(* Logix 5000 project; controller L3 vendor 1 type 14 code 92 rev 20.12; software revision 20.04; part 8 of 9 *)
(* tags used below, declared in another part *)
   A_CV_COLMAT : REAL;
   aux_spano : DINT;
   B3 : DINT[100];
   CONV_PID_N10_130 : PID;   // *** Tag created for conversion to PID type required for instruction translation ***
   CSG_N_VENTILO : REAL;
   CV_ANO : REAL;
   dif_I_red : DINT;
   F8 : REAL[100];
   inc_ano : DINT;
   khighano : DINT;
   klowano : DINT;
   L3_stat : DINT[20];
   limBBtano : DINT;
   limBtano : DINT;
   limhhtano : DINT;
   limhtano : DINT;
   M_nbr_ventilo_ano : DINT;
   mem_i_tot : DINT;
   N10 : DINT[233];
   N7 : DINT[200];
   N9 : DINT[200];   // niveau decapage vers lancy (n9[10) ;;N9[70]
   NCOM : INT[20];
   offsetano : DINT;
   offsetano_tdesc : DINT;
   offsetano_Tup : DINT;
   par_p1_ano : DINT;
   par_p2_ano : DINT;
   par_p3_ano : DINT;
   par_p4_ano : DINT;
   par_p5_ano : DINT;
   par_p6_ano : DINT;
   pid_ANO : PID;
   pid_colmat : PID;
   PIDwkk : PID;
   s_bp_neutral : BOOL;
   s_bp_stop_acide : BOOL;
   s_bp_strt_acide : BOOL;
   s_csg_ventilo_ano : DINT;
   s_nbr_ventilo_ano : DINT;
   S_Q_DEM_h2so4 : DINT;
   S_SP_ANO : DINT;
   S_T_ANO : DINT;
   SCP_CV_ANO : SCP;
   SCP_CV_COLMAT : SCP;
   SCP_CV_VENTILO : SCP;
   stat_L3 : DINT[20];
   T4 : TIMER[180];
   wkk_L3 : DINT[125];
(* _2_GENERAL, continued *)

ROUTINE _5_ACIDE   (* ladder *)
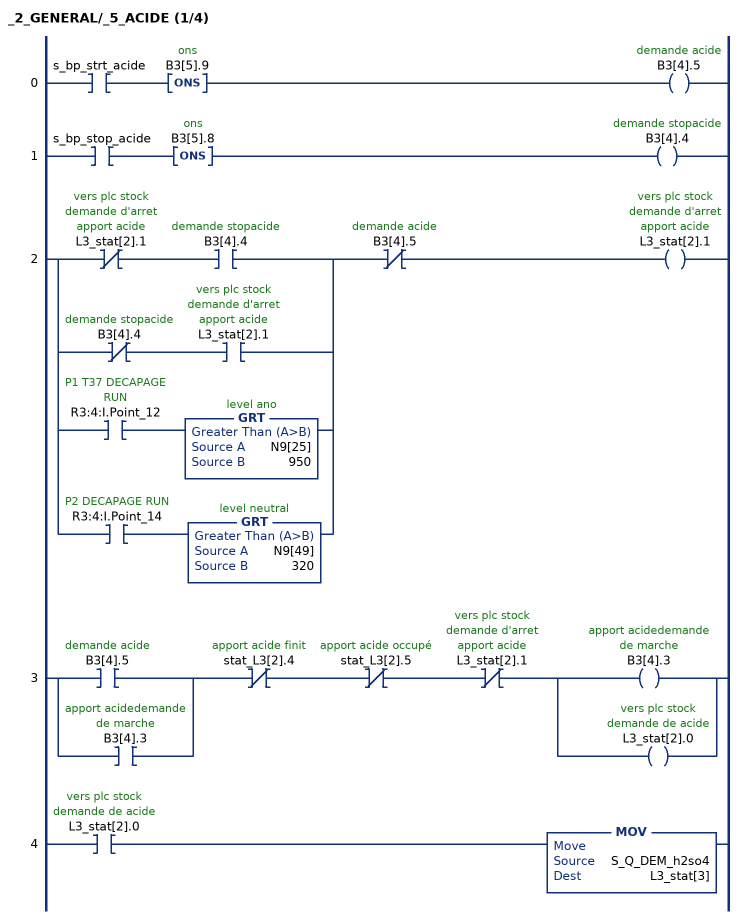
   0: XIC(s_bp_strt_acide)ONS(B3[5].9)OTE(B3[4].5);
   1: XIC(s_bp_stop_acide)ONS(B3[5].8)OTE(B3[4].4);
   2: [XIO(L3_stat[2].1) XIC(B3[4].4) ,XIO(B3[4].4) XIC(L3_stat[2].1) ,XIC(R3:4:I.Point_12) GRT(N9[25],950) ,XIC(R3:4:I.Point_14) GRT(N9[49],320) ]XIO(B3[4].5)OTE(L3_stat[2].1);
   3: [XIC(B3[4].5) ,XIC(B3[4].3) ]XIO(stat_L3[2].4)XIO(stat_L3[2].5)XIO(L3_stat[2].1)[OTE(B3[4].3) ,OTE(L3_stat[2].0) ];
   4: XIC(L3_stat[2].0)MOV(S_Q_DEM_h2so4,L3_stat[3]);
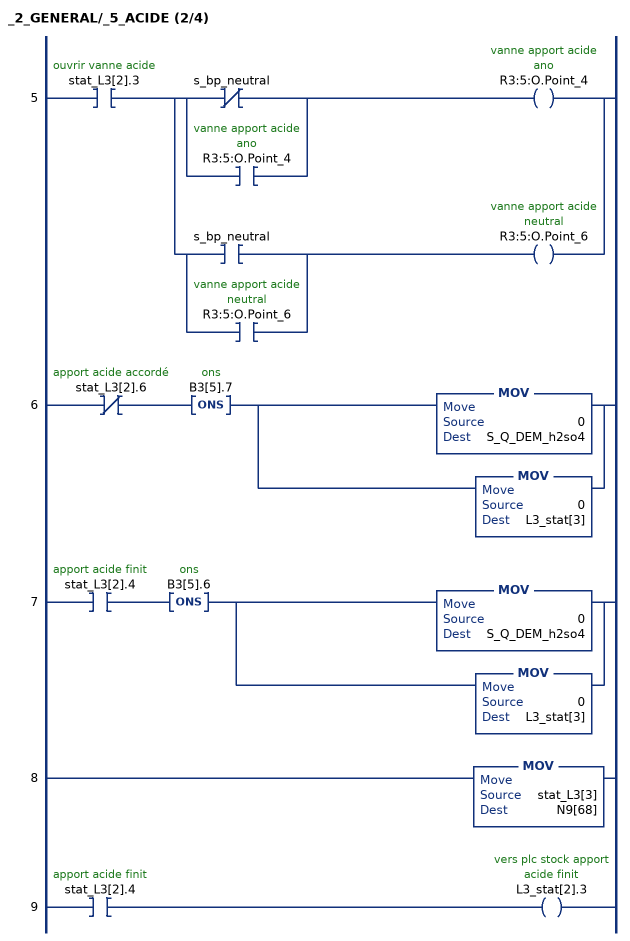
   5: XIC(stat_L3[2].3)[[XIO(s_bp_neutral) ,XIC(R3:5:O.Point_4) ] OTE(R3:5:O.Point_4) ,[XIC(s_bp_neutral) ,XIC(R3:5:O.Point_6) ] OTE(R3:5:O.Point_6) ];
   6: XIO(stat_L3[2].6)ONS(B3[5].7)[MOV(0,S_Q_DEM_h2so4) ,MOV(0,L3_stat[3]) ];
   7: XIC(stat_L3[2].4)ONS(B3[5].6)[MOV(0,S_Q_DEM_h2so4) ,MOV(0,L3_stat[3]) ];
   8: MOV(stat_L3[3],N9[68]);
   9: XIC(stat_L3[2].4)OTE(L3_stat[2].3);
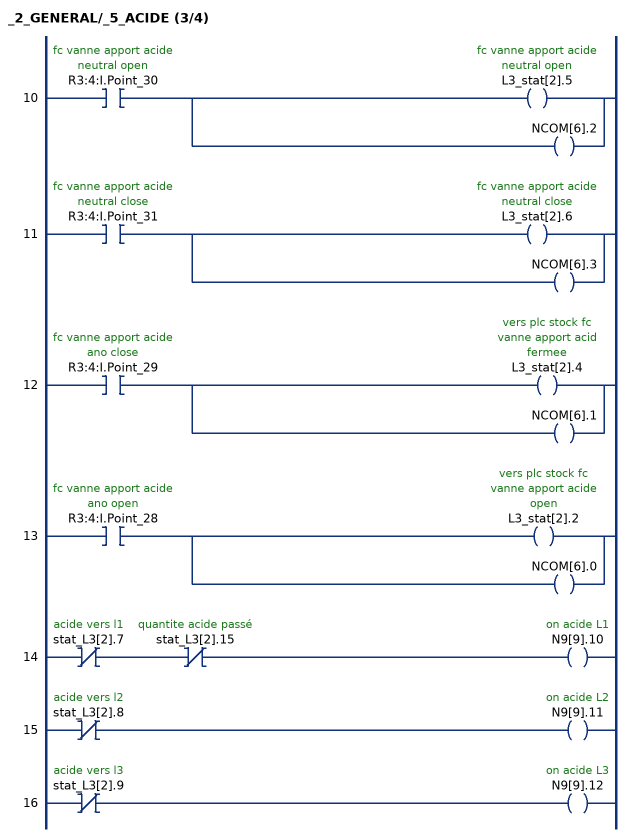
   10: XIC(R3:4:I.Point_30)[OTE(L3_stat[2].5) ,OTE(NCOM[6].2) ];
   11: XIC(R3:4:I.Point_31)[OTE(L3_stat[2].6) ,OTE(NCOM[6].3) ];
   12: XIC(R3:4:I.Point_29)[OTE(L3_stat[2].4) ,OTE(NCOM[6].1) ];
   13: XIC(R3:4:I.Point_28)[OTE(L3_stat[2].2) ,OTE(NCOM[6].0) ];
   14: XIO(stat_L3[2].7)XIO(stat_L3[2].15)OTE(N9[9].10);
   15: XIO(stat_L3[2].8)OTE(N9[9].11);
   16: XIO(stat_L3[2].9)OTE(N9[9].12);
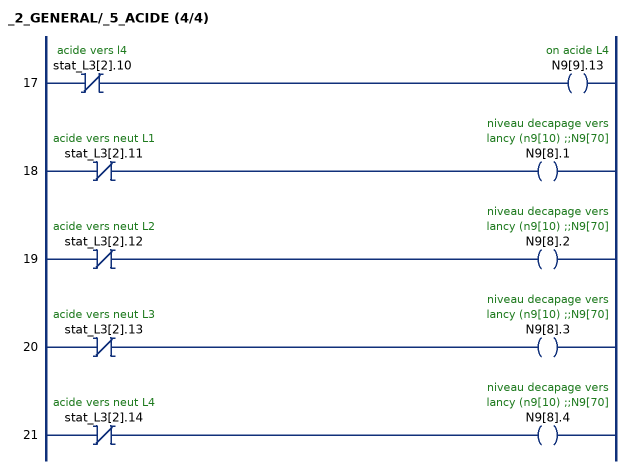
   17: XIO(stat_L3[2].10)OTE(N9[9].13);
   18: XIO(stat_L3[2].11)OTE(N9[8].1);
   19: XIO(stat_L3[2].12)OTE(N9[8].2);
   20: XIO(stat_L3[2].13)OTE(N9[8].3);
   21: XIO(stat_L3[2].14)OTE(N9[8].4);
END_ROUTINE

ROUTINE _6_REG_T_COL   (* ladder *)
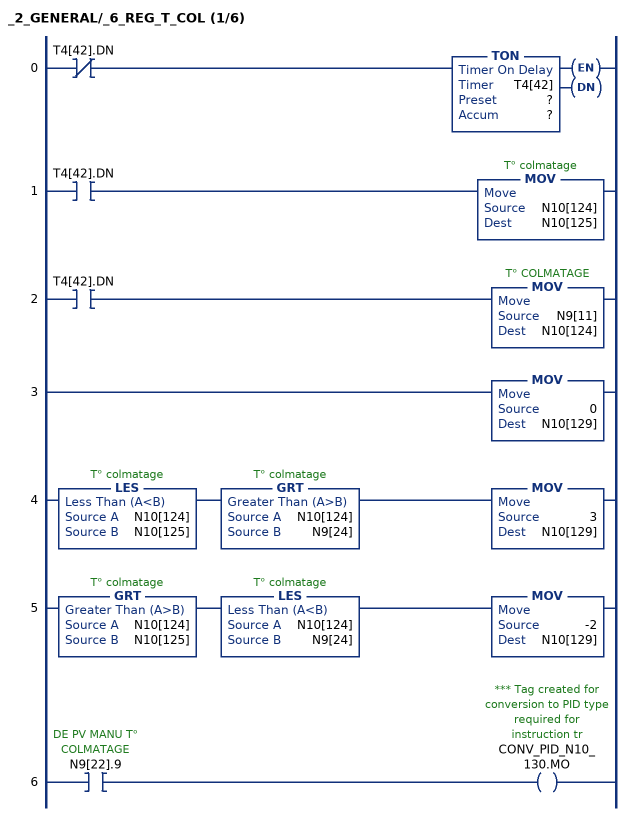
   0: XIO(T4[42].DN)TON(T4[42],?,?);
   1: XIC(T4[42].DN)MOV(N10[124],N10[125]);
   2: XIC(T4[42].DN)MOV(N9[11],N10[124]);
   3: MOV(0,N10[129]);
   4: LES(N10[124],N10[125])GRT(N10[124],N9[24])MOV(3,N10[129]);
   5: GRT(N10[124],N10[125])LES(N10[124],N9[24])MOV(-2,N10[129]);
   6: XIC(N9[22].9)OTE(CONV_PID_N10_130.MO);
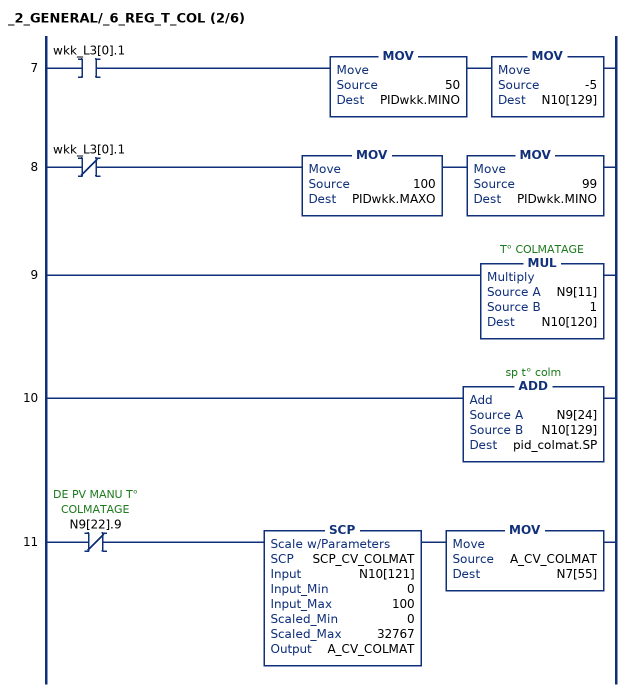
   7: XIC(wkk_L3[0].1)MOV(50,PIDwkk.MINO)MOV(-5,N10[129]);
   8: XIO(wkk_L3[0].1)MOV(100,PIDwkk.MAXO)MOV(99,PIDwkk.MINO);
   9: MUL(N9[11],1,N10[120]);
   10: ADD(N9[24],N10[129],pid_colmat.SP);
   11: XIO(N9[22].9)SCP(SCP_CV_COLMAT,N10[121],0,100,0,32767,A_CV_COLMAT)MOV(A_CV_COLMAT,N7[55]);
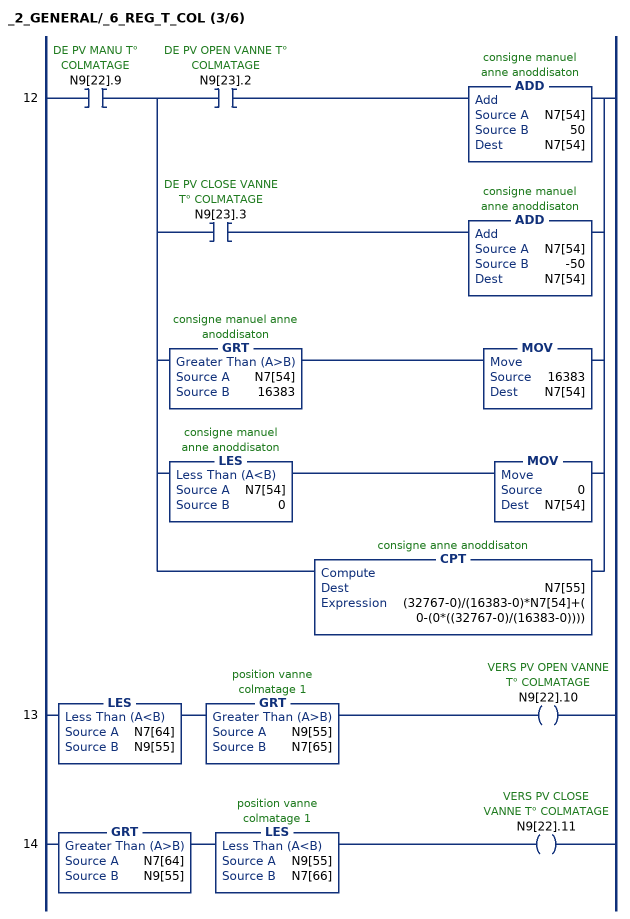
   12: XIC(N9[22].9)[XIC(N9[23].2) ADD(N7[54],50,N7[54]) ,XIC(N9[23].3) ADD(N7[54],-50,N7[54]) ,GRT(N7[54],16383) MOV(16383,N7[54]) ,LES(N7[54],0) MOV(0,N7[54]) ,CPT(N7[55],(32767-0)/(16383-0)*N7[54]+(0-(0*((32767-0)/(16383-0))))) ];
   13: LES(N7[64],N9[55])GRT(N9[55],N7[65])OTE(N9[22].10);
   14: GRT(N7[64],N9[55])LES(N9[55],N7[66])OTE(N9[22].11);
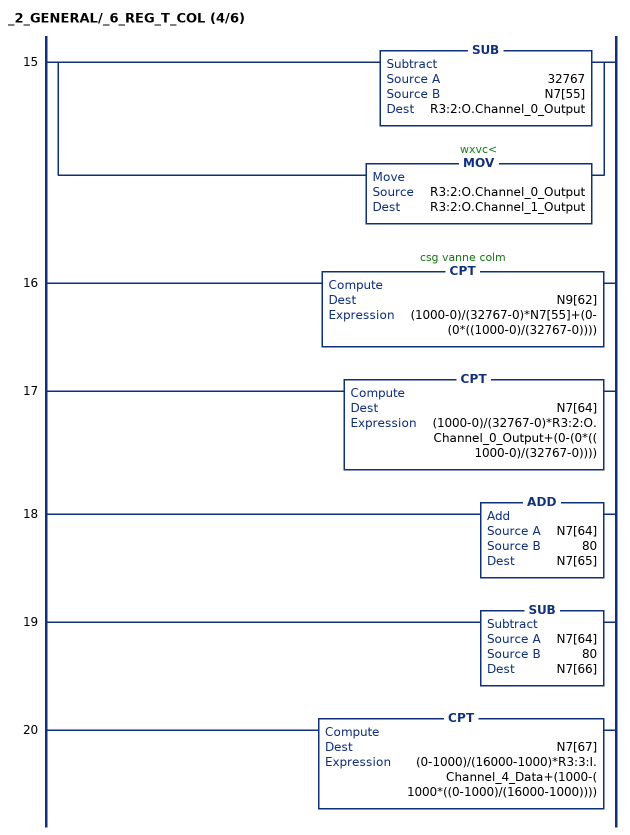
   15: [SUB(32767,N7[55],R3:2:O.Channel_0_Output) ,MOV(R3:2:O.Channel_0_Output,R3:2:O.Channel_1_Output) ];
   16: CPT(N9[62],(1000-0)/(32767-0)*N7[55]+(0-(0*((1000-0)/(32767-0)))));
   17: CPT(N7[64],(1000-0)/(32767-0)*R3:2:O.Channel_0_Output+(0-(0*((1000-0)/(32767-0)))));
   18: ADD(N7[64],80,N7[65]);
   19: SUB(N7[64],80,N7[66]);
   20: CPT(N7[67],(0-1000)/(16000-1000)*R3:3:I.Channel_4_Data+(1000-(1000*((0-1000)/(16000-1000)))));
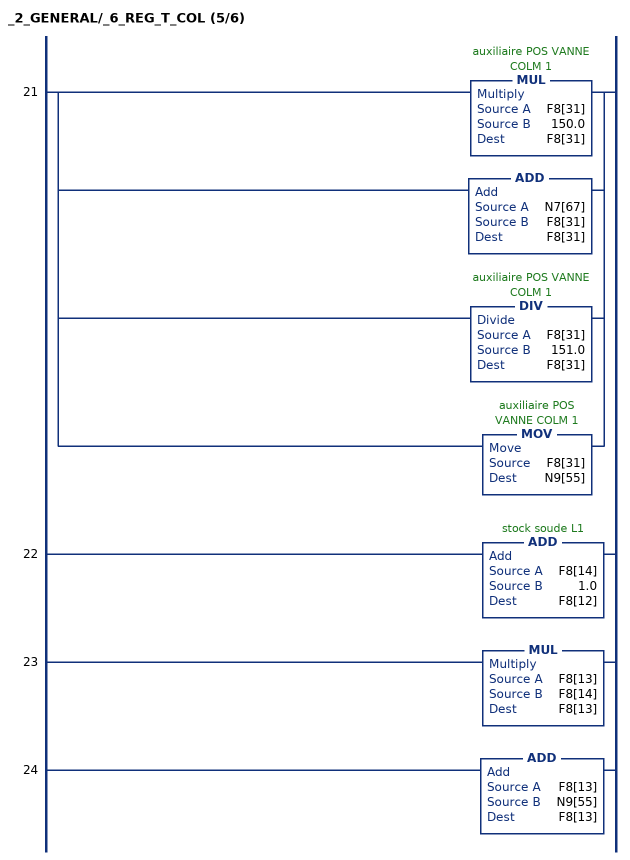
   21: [MUL(F8[31],150.0,F8[31]) ,ADD(N7[67],F8[31],F8[31]) ,DIV(F8[31],151.0,F8[31]) ,MOV(F8[31],N9[55]) ];
   22: ADD(F8[14],1.0,F8[12]);
   23: MUL(F8[13],F8[14],F8[13]);
   24: ADD(F8[13],N9[55],F8[13]);
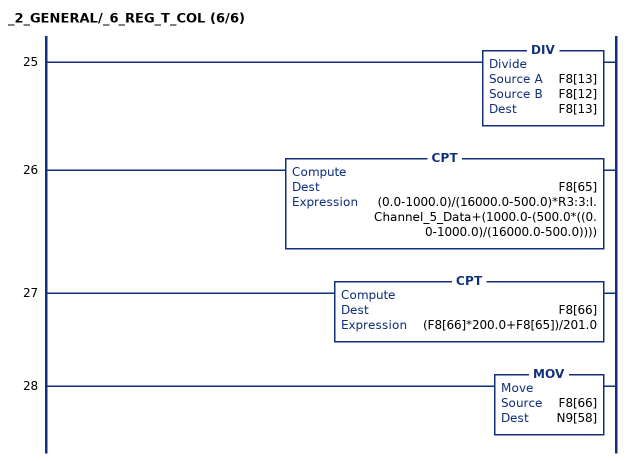
   25: DIV(F8[13],F8[12],F8[13]);
   26: CPT(F8[65],(0.0-1000.0)/(16000.0-500.0)*R3:3:I.Channel_5_Data+(1000.0-(500.0*((0.0-1000.0)/(16000.0-500.0)))));
   27: CPT(F8[66],(F8[66]*200.0+F8[65])/201.0);
   28: MOV(F8[66],N9[58]);
END_ROUTINE

ROUTINE _9_regul_ano   (* ladder *)
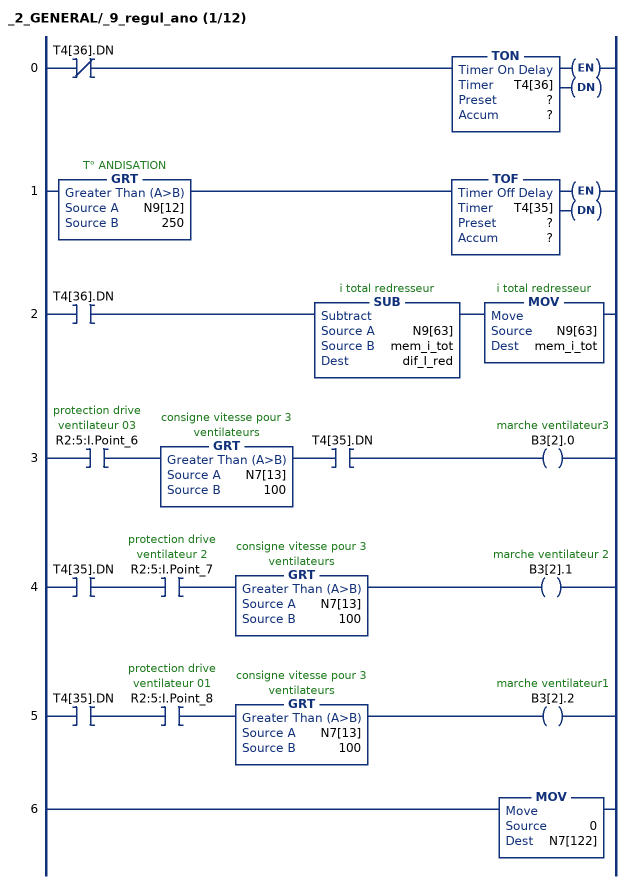
   0: XIO(T4[36].DN)TON(T4[36],?,?);
   1: GRT(N9[12],250)TOF(T4[35],?,?);
   2: XIC(T4[36].DN)SUB(N9[63],mem_i_tot,dif_I_red)MOV(N9[63],mem_i_tot);
   3: XIC(R2:5:I.Point_6)GRT(N7[13],100)XIC(T4[35].DN)OTE(B3[2].0);
   4: XIC(T4[35].DN)XIC(R2:5:I.Point_7)GRT(N7[13],100)OTE(B3[2].1);
   5: XIC(T4[35].DN)XIC(R2:5:I.Point_8)GRT(N7[13],100)OTE(B3[2].2);
   6: MOV(0,N7[122]);
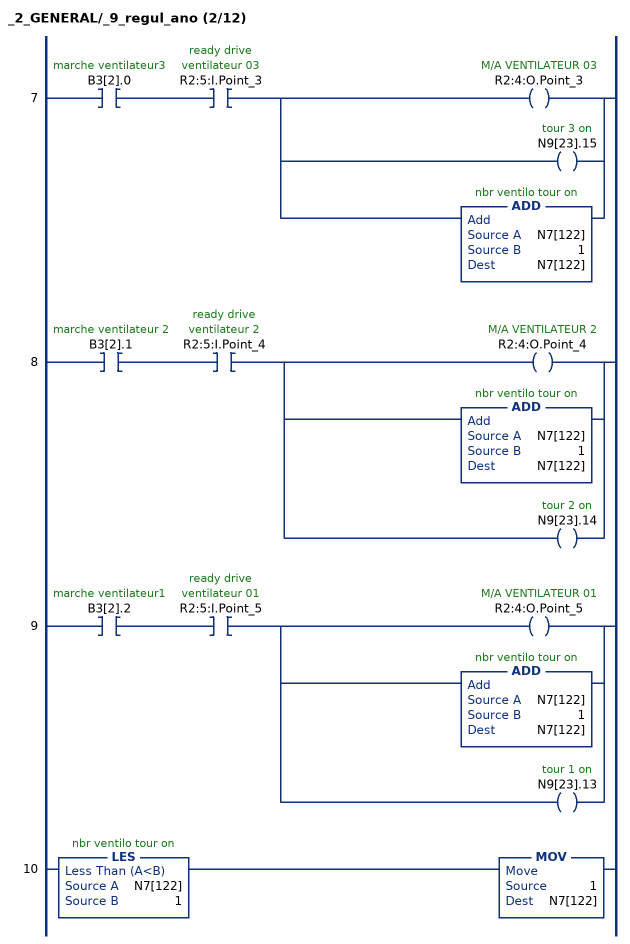
   7: XIC(B3[2].0)XIC(R2:5:I.Point_3)[OTE(R2:4:O.Point_3) ,OTE(N9[23].15) ,ADD(N7[122],1,N7[122]) ];
   8: XIC(B3[2].1)XIC(R2:5:I.Point_4)[OTE(R2:4:O.Point_4) ,ADD(N7[122],1,N7[122]) ,OTE(N9[23].14) ];
   9: XIC(B3[2].2)XIC(R2:5:I.Point_5)[OTE(R2:4:O.Point_5) ,ADD(N7[122],1,N7[122]) ,OTE(N9[23].13) ];
   10: LES(N7[122],1)MOV(1,N7[122]);
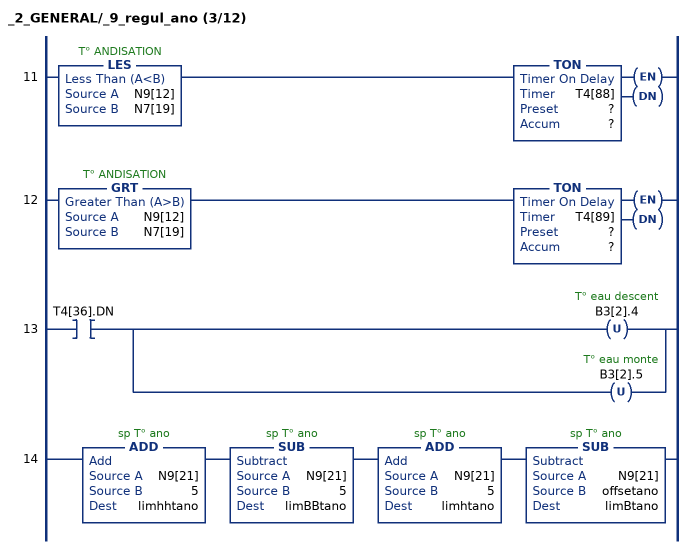
   11: LES(N9[12],N7[19])TON(T4[88],?,?);
   12: GRT(N9[12],N7[19])TON(T4[89],?,?);
   13: XIC(T4[36].DN)[OTU(B3[2].4) ,OTU(B3[2].5) ];
   14: ADD(N9[21],5,limhhtano)SUB(N9[21],5,limBBtano)ADD(N9[21],5,limhtano)SUB(N9[21],offsetano,limBtano);
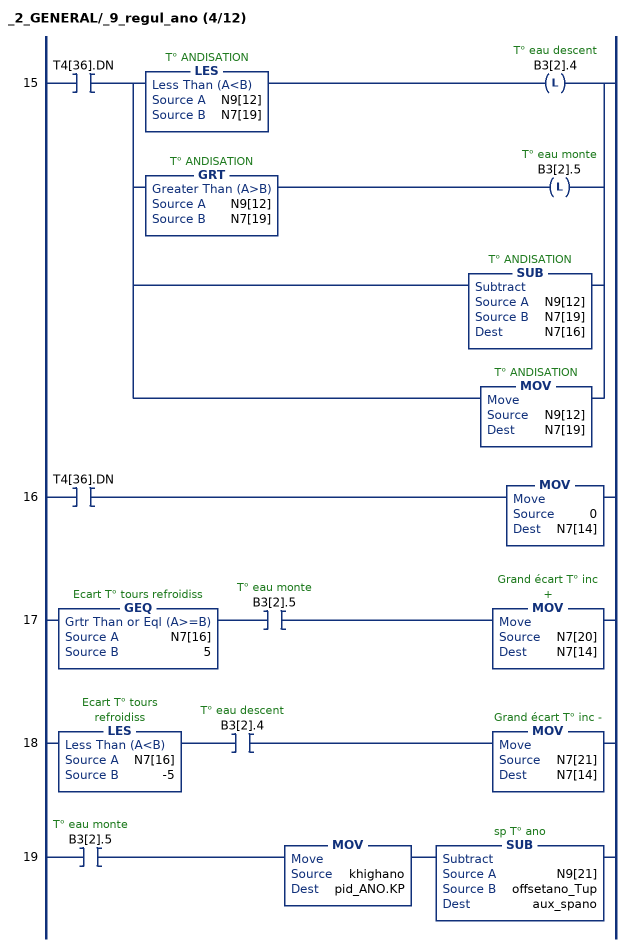
   15: XIC(T4[36].DN)[LES(N9[12],N7[19]) OTL(B3[2].4) ,GRT(N9[12],N7[19]) OTL(B3[2].5) ,SUB(N9[12],N7[19],N7[16]) ,MOV(N9[12],N7[19]) ];
   16: XIC(T4[36].DN)MOV(0,N7[14]);
   17: GEQ(N7[16],5)XIC(B3[2].5)MOV(N7[20],N7[14]);
   18: LES(N7[16],-5)XIC(B3[2].4)MOV(N7[21],N7[14]);
   19: XIC(B3[2].5)MOV(khighano,pid_ANO.KP)SUB(N9[21],offsetano_Tup,aux_spano);
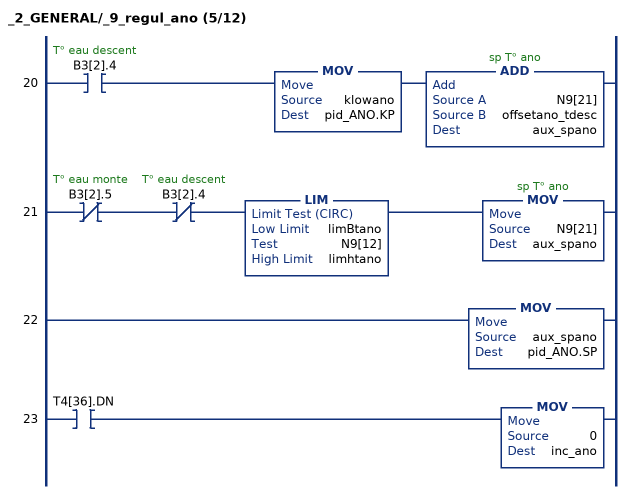
   20: XIC(B3[2].4)MOV(klowano,pid_ANO.KP)ADD(N9[21],offsetano_tdesc,aux_spano);
   21: XIO(B3[2].5)XIO(B3[2].4)LIM(limBtano,N9[12],limhtano)MOV(N9[21],aux_spano);
   22: MOV(aux_spano,pid_ANO.SP);
   23: XIC(T4[36].DN)MOV(0,inc_ano);
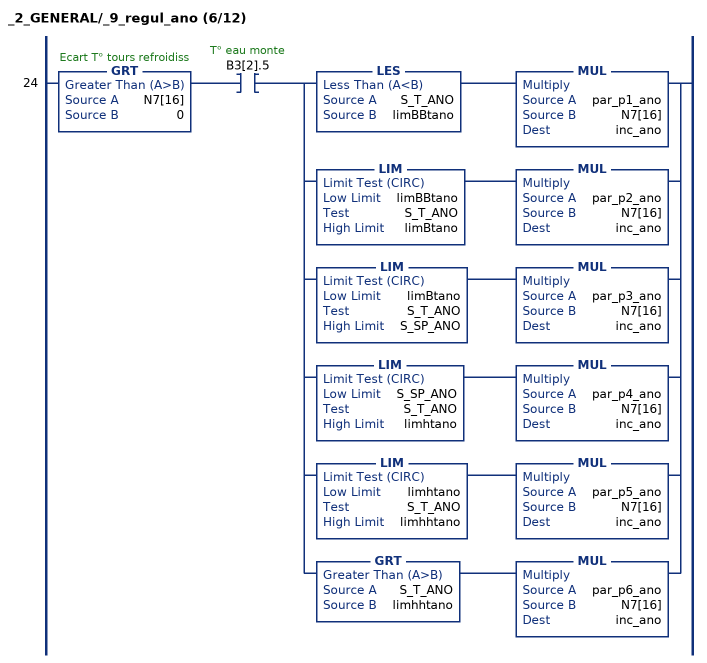
   24: GRT(N7[16],0)XIC(B3[2].5)[LES(S_T_ANO,limBBtano) MUL(par_p1_ano,N7[16],inc_ano) ,LIM(limBBtano,S_T_ANO,limBtano) MUL(par_p2_ano,N7[16],inc_ano) ,LIM(limBtano,S_T_ANO,S_SP_ANO) MUL(par_p3_ano,N7[16],inc_ano) ,LIM(S_SP_ANO,S_T_ANO,limhtano) MUL(par_p4_ano,N7[16],inc_ano) ,LIM(limhtano,S_T_ANO,limhhtano) MUL(par_p5_ano,N7[16],inc_ano) ,GRT(S_T_ANO,limhhtano) MUL(par_p6_ano,N7[16],inc_ano) ];
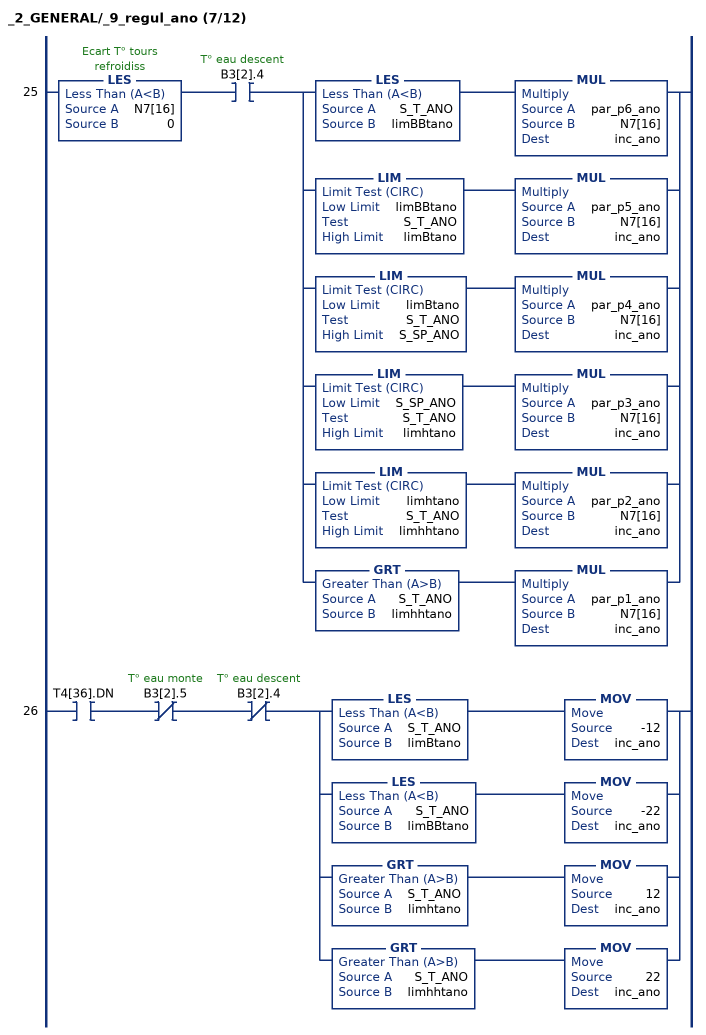
   25: LES(N7[16],0)XIC(B3[2].4)[LES(S_T_ANO,limBBtano) MUL(par_p6_ano,N7[16],inc_ano) ,LIM(limBBtano,S_T_ANO,limBtano) MUL(par_p5_ano,N7[16],inc_ano) ,LIM(limBtano,S_T_ANO,S_SP_ANO) MUL(par_p4_ano,N7[16],inc_ano) ,LIM(S_SP_ANO,S_T_ANO,limhtano) MUL(par_p3_ano,N7[16],inc_ano) ,LIM(limhtano,S_T_ANO,limhhtano) MUL(par_p2_ano,N7[16],inc_ano) ,GRT(S_T_ANO,limhhtano) MUL(par_p1_ano,N7[16],inc_ano) ];
   26: XIC(T4[36].DN)XIO(B3[2].5)XIO(B3[2].4)[LES(S_T_ANO,limBtano) MOV(-12,inc_ano) ,LES(S_T_ANO,limBBtano) MOV(-22,inc_ano) ,GRT(S_T_ANO,limhtano) MOV(12,inc_ano) ,GRT(S_T_ANO,limhhtano) MOV(22,inc_ano) ];
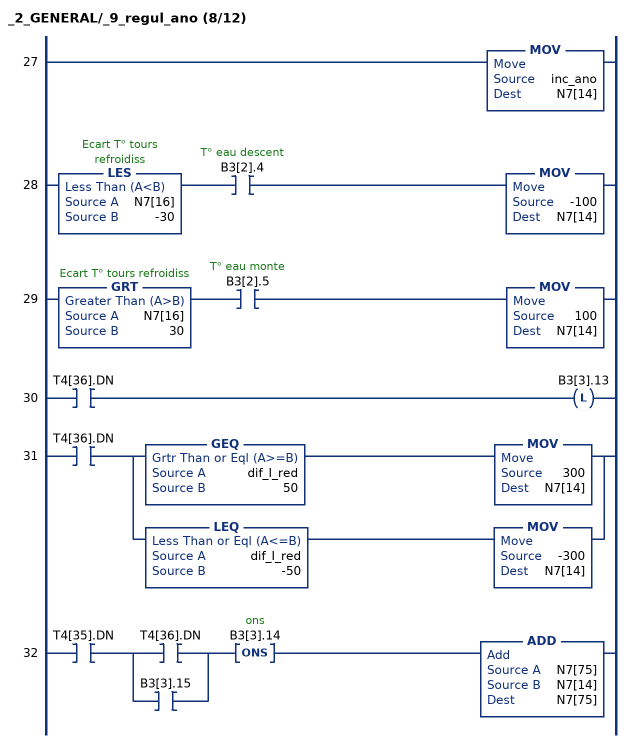
   27: MOV(inc_ano,N7[14]);
   28: LES(N7[16],-30)XIC(B3[2].4)MOV(-100,N7[14]);
   29: GRT(N7[16],30)XIC(B3[2].5)MOV(100,N7[14]);
   30: XIC(T4[36].DN)OTL(B3[3].13);
   31: XIC(T4[36].DN)[GEQ(dif_I_red,50) MOV(300,N7[14]) ,LEQ(dif_I_red,-50) MOV(-300,N7[14]) ];
   32: XIC(T4[35].DN)[XIC(T4[36].DN) ,XIC(B3[3].15) ]ONS(B3[3].14)ADD(N7[75],N7[14],N7[75]);
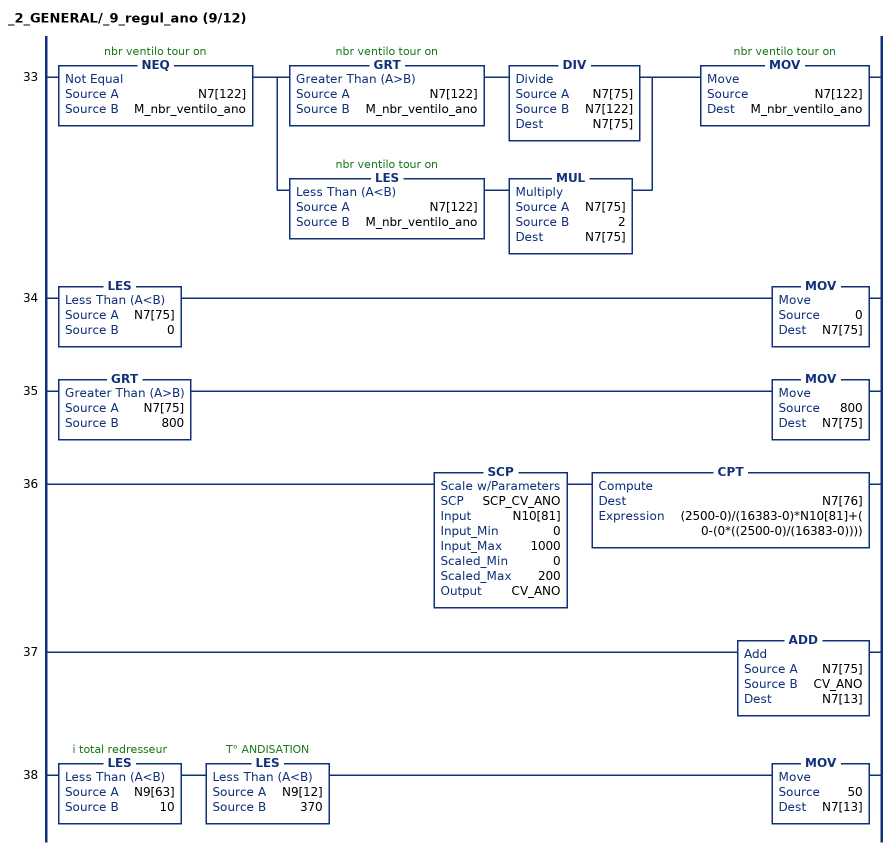
   33: NEQ(N7[122],M_nbr_ventilo_ano)[GRT(N7[122],M_nbr_ventilo_ano) DIV(N7[75],N7[122],N7[75]) ,LES(N7[122],M_nbr_ventilo_ano) MUL(N7[75],2,N7[75]) ]MOV(N7[122],M_nbr_ventilo_ano);
   34: LES(N7[75],0)MOV(0,N7[75]);
   35: GRT(N7[75],800)MOV(800,N7[75]);
   36: SCP(SCP_CV_ANO,N10[81],0,1000,0,200,CV_ANO)CPT(N7[76],(2500-0)/(16383-0)*N10[81]+(0-(0*((2500-0)/(16383-0)))));
   37: ADD(N7[75],CV_ANO,N7[13]);
   38: LES(N9[63],10)LES(N9[12],370)MOV(50,N7[13]);
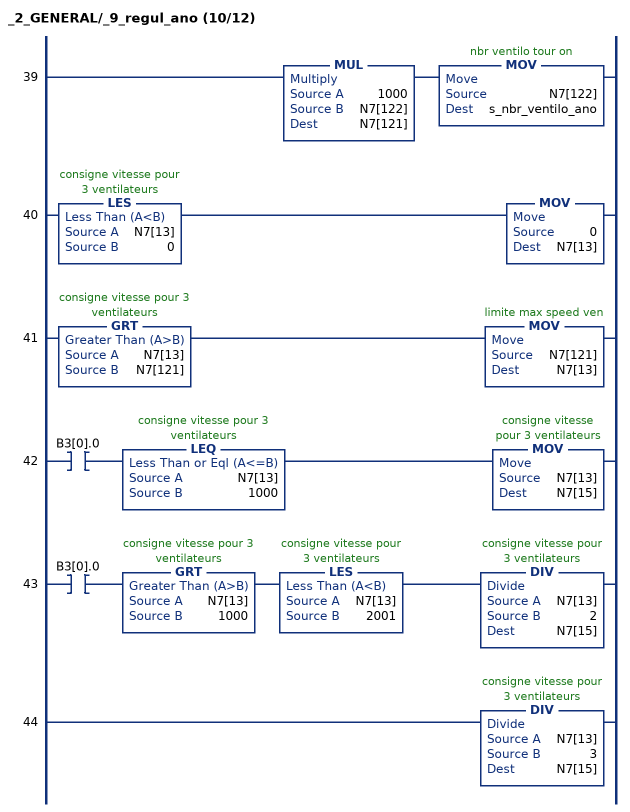
   39: MUL(1000,N7[122],N7[121])MOV(N7[122],s_nbr_ventilo_ano);
   40: LES(N7[13],0)MOV(0,N7[13]);
   41: GRT(N7[13],N7[121])MOV(N7[121],N7[13]);
   42: XIC(B3[0].0)LEQ(N7[13],1000)MOV(N7[13],N7[15]);
   43: XIC(B3[0].0)GRT(N7[13],1000)LES(N7[13],2001)DIV(N7[13],2,N7[15]);
   44: DIV(N7[13],3,N7[15]);
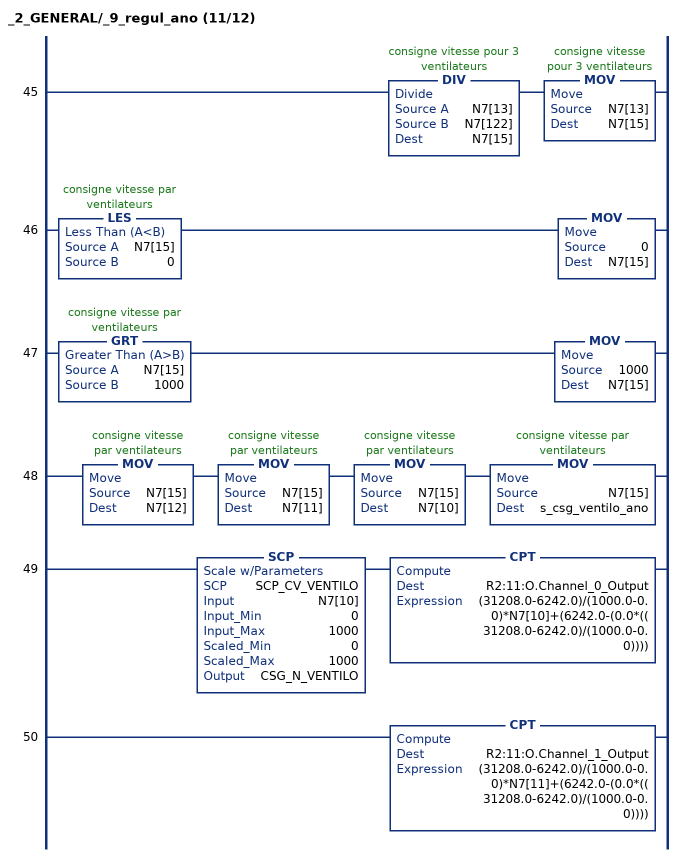
   45: DIV(N7[13],N7[122],N7[15])MOV(N7[13],N7[15]);
   46: LES(N7[15],0)MOV(0,N7[15]);
   47: GRT(N7[15],1000)MOV(1000,N7[15]);
   48: MOV(N7[15],N7[12])MOV(N7[15],N7[11])MOV(N7[15],N7[10])MOV(N7[15],s_csg_ventilo_ano);
   49: SCP(SCP_CV_VENTILO,N7[10],0,1000,0,1000,CSG_N_VENTILO)CPT(R2:11:O.Channel_0_Output,(31208.0-6242.0)/(1000.0-0.0)*N7[10]+(6242.0-(0.0*((31208.0-6242.0)/(1000.0-0.0)))));
   50: CPT(R2:11:O.Channel_1_Output,(31208.0-6242.0)/(1000.0-0.0)*N7[11]+(6242.0-(0.0*((31208.0-6242.0)/(1000.0-0.0)))));
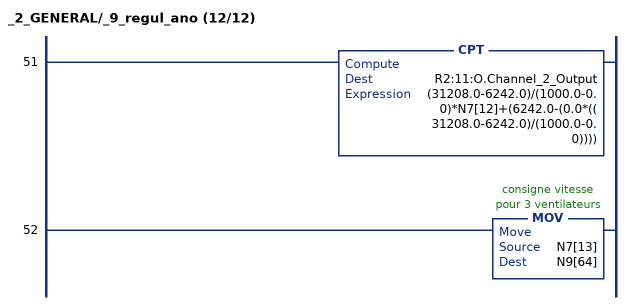
   51: CPT(R2:11:O.Channel_2_Output,(31208.0-6242.0)/(1000.0-0.0)*N7[12]+(6242.0-(0.0*((31208.0-6242.0)/(1000.0-0.0)))));
   52: MOV(N7[13],N9[64]);
END_ROUTINE
